Staubli VAL3: FCheckInBox2Pos.pgx

public program FCheckInBox2Pos(tool t_tool, frame fr_frame, bool& b_inArea[], bool& x_bJtEnabCheck[], bool& x_bPosEnabCheck[], num& x_nRobCtrlJts[], num& x_nRobCtrlArea[])
// Pruefen ob Roboter innerhalb eines definierten Bereichs
  local trsf tr_here
  local point p_here
  local trsf tr_NegPos
  local trsf tr_PosPos
  local trsf tr_BoxPos1
  local trsf tr_BoxPos2
  local jointRx j_here
  local num i
  local num l_nItem[6]
begin
  //Header
  if false
    //判断机器人是否属于所设定的空间盒子中
    //Parameter:
    //  p_BoxPos1: Position 1 (包括开始位置跟结束位置)
    //  p_BoxPos2: Position 2 (包括开始位置跟结束位置)
    //  b_inArea: 返回参数  true  : 机器人在矩形中
    //                          false : 机器人属于非矩形中
    //
  endIf
  //判断变量返回
  b_inArea=true
  p_here=here(t_tool,fr_frame)
  j_here=herej()
  ///////////////////////////////////////////////////
  tr_here=p_here.trsf
  l_nItem[0]=j_here.j1
  l_nItem[1]=j_here.j2
  l_nItem[2]=j_here.j3
  l_nItem[3]=j_here.j4
  l_nItem[4]=j_here.j5
  l_nItem[5]=j_here.j6
  for i=0 to 5
    if x_bJtEnabCheck[i]
      if l_nItem[i]>=x_nRobCtrlJts[i*2+1] or l_nItem[i]<=x_nRobCtrlJts[i*2]
        b_inArea=false
      endIf
    endIf
  endFor
  /////////////////////////////////////////
  l_nItem[0]=p_here.trsf.x
  l_nItem[1]=p_here.trsf.y
  l_nItem[2]=p_here.trsf.z
  l_nItem[3]=p_here.trsf.rx
  l_nItem[4]=p_here.trsf.ry
  l_nItem[5]=p_here.trsf.rz
  for i=0 to 5
    if x_bPosEnabCheck[i]
      if l_nItem[i]>=x_nRobCtrlArea[i*2+1] or l_nItem[i]<=x_nRobCtrlArea[i*2]
        b_inArea=false
      endIf
    endIf
  endFor
end
